// TwinCAT 3 PLC project Plc_Ampel
// ProgramVersion: 3.1.4023.0
// libraries:
//   Tc2_Standard, * (Beckhoff Automation GmbH)
//   Tc2_System, * (Beckhoff Automation GmbH)
//   Tc3_Module, * (Beckhoff Automation GmbH)
//   VisuSymbols,3.5.10.0,System
// project tree:
//   DUTs/ EN_TRAFFICLIGHT_STATE.TcDUT
//   / GlobalTextList.TcGTLO, PlcTask.TcTTO, Visualization Manager.TcVMO (not stored)
//   POUs/ MAIN.TcPOU, FB_TrafficLight.TcPOU
//   VISUs/ VISU_TrafficLight.TcVIS
// (motion and I/O tree: see PLC project plc_safe)
// real-time tasks:
//   TASK PlcTask: cycle T#10ms, priority 20, ADS port 350
//   TASK PlcTask1: cycle T#10ms, priority 21, ADS port 351

CONFIGURATION Plc_Ampel
    RESOURCE PLC ON TwinCAT3
        TASK PlcTask(INTERVAL := T#10ms, PRIORITY := 21);
        PROGRAM MAIN WITH PlcTask : MAIN;
    END_RESOURCE
END_CONFIGURATION

// ---- DUTs/EN_TRAFFICLIGHT_STATE.TcDUT
{attribute 'qualified_only'}
{attribute 'strict'}
TYPE EN_TRAFFICLIGHT_STATE :
(
	STATE_UNDEFINED := 0,
	STATE_INIT,
	STATE_DISABLED,
	STATE_RED,
	STATE_RED_YELLOW,
	STATE_YELLOW,
	STATE_GREEN
);
END_TYPE

// ---- POUs/MAIN.TcPOU
PROGRAM MAIN
VAR
	trafficLight_1			: FB_TrafficLight;
	
	// control variables
	clear					: BOOL;
	block					: BOOL;
	disable					: BOOL;
	
	// output variables
	red						: BOOL;
	yellow					: BOOL;
	green					: BOOL;
END_VAR

trafficLight_1(clear_road := clear, block_road := block, disable_system := disable);

red := trafficLight_1.red_light;
yellow := trafficLight_1.yellow_light;
green := trafficLight_1.green_light;

END_PROGRAM

// ---- POUs/FB_TrafficLight.TcPOU
FUNCTION_BLOCK FB_TrafficLight
VAR_INPUT
	clear_road 			: BOOL;
	block_road 			: BOOL;
	disable_system		: BOOL;
END_VAR
VAR_OUTPUT
	red_light			: BOOL;
	yellow_light		: BOOL;
	green_light			: BOOL;
END_VAR
VAR
	// state variables
	currentState		: 	EN_TRAFFICLIGHT_STATE := EN_TRAFFICLIGHT_STATE.STATE_INIT;
	lastState			: 	EN_TRAFFICLIGHT_STATE := EN_TRAFFICLIGHT_STATE.STATE_UNDEFINED;
	timer				: 	TON;
	// flag to reset the timer after the state machine has used it
	resetTimer			:	BOOL;
	// flag to update last state
	transitionDone		: 	BOOL;
END_VAR

timer();  // call timer

// state machine
CASE currentState OF
	EN_TRAFFICLIGHT_STATE.STATE_UNDEFINED:
	// jump to init	
	currentState := EN_TRAFFICLIGHT_STATE.STATE_INIT;
	
	//*****************************//
	EN_TRAFFICLIGHT_STATE.STATE_INIT:
	// jump to red
	currentState := EN_TRAFFICLIGHT_STATE.STATE_RED;
	
	//*****************************//
	EN_TRAFFICLIGHT_STATE.STATE_RED:
	// entry action
	IF(currentState <> lastState) THEN
		// enable only red light
		red_light := TRUE; yellow_light := FALSE; green_light := FALSE;
		lastState := currentState;  // update last state
	END_IF
	
	// clear road (prio 2)
	IF(clear_road) THEN
		currentState := EN_TRAFFICLIGHT_STATE.STATE_RED_YELLOW;
	END_IF
	
	// clear road (prio 1)
	IF(disable_system) THEN
		currentState := EN_TRAFFICLIGHT_STATE.STATE_DISABLED;
	END_IF
	
	//*****************************//
	EN_TRAFFICLIGHT_STATE.STATE_RED_YELLOW:
	// entry action
	IF(currentState <> lastState) THEN
		// enable red and yellow light
		red_light := TRUE; yellow_light := TRUE; green_light := FALSE;
		lastState := currentState;  // update last state
	END_IF
	
	// start timer for automatic state change
	timer.PT := T#2S;
	timer.IN := TRUE;
	
	// timer finished => exit action
	IF timer.Q THEN
		currentState := EN_TRAFFICLIGHT_STATE.STATE_GREEN;
		resetTimer := TRUE;
	END_IF
	
	//*****************************//
	EN_TRAFFICLIGHT_STATE.STATE_YELLOW:
	// entry action
	IF(currentState <> lastState) THEN
		// enable yellow light only
		red_light := FALSE; yellow_light := TRUE; green_light := FALSE;
		lastState := currentState;  // update last state
	END_IF
	
	// start timer for automatic state change
	timer.PT := T#5S;
	timer.IN := TRUE;
	
	// timer finished => exit action
	IF timer.Q THEN
		currentState := EN_TRAFFICLIGHT_STATE.STATE_RED;
		resetTimer := TRUE;
	END_IF
	
	//*****************************//
	EN_TRAFFICLIGHT_STATE.STATE_GREEN:
	// entry action
	IF(currentState <> lastState) THEN
		// enable green light only
		red_light := FALSE; yellow_light := FALSE; green_light := TRUE;
		lastState := currentState;  // update last state
	END_IF
	
	// block_road signal
	IF(block_road) THEN
		currentState := EN_TRAFFICLIGHT_STATE.STATE_YELLOW;
	END_IF
	
	//*****************************//
	EN_TRAFFICLIGHT_STATE.STATE_DISABLED:
	// disable all lights
	red_light := FALSE; green_light := FALSE;
	
	// start timer for yellow blinking
	timer.PT := T#1S;
	timer.IN := TRUE;
	
	// invert yellow light (blink)
	IF timer.Q THEN
		yellow_light := NOT yellow_light;
		resetTimer := TRUE;
	END_IF
	
	// system was re-enabled 
	IF (disable_system = FALSE) THEN
		lastState := currentState;  // update last state
		currentState := EN_TRAFFICLIGHT_STATE.STATE_RED;
		resetTimer := TRUE;
	END_IF
	
END_CASE

// reset timer since it was used
IF resetTimer THEN
	timer.IN := FALSE;
	timer();  // call to trigger edge
	resetTimer := FALSE;	
END_IF

END_FUNCTION_BLOCK

// ---- GlobalTextList.TcGTLO
TEXTLIST GlobalTextList
  241 = 'Block road'
  918 = 'Clear road'
  437 = 'Control'
  462 = 'Disable system'
  422 = 'Traffic Light'
END_TEXTLIST

// ---- VISUs/VISU_TrafficLight.TcVIS
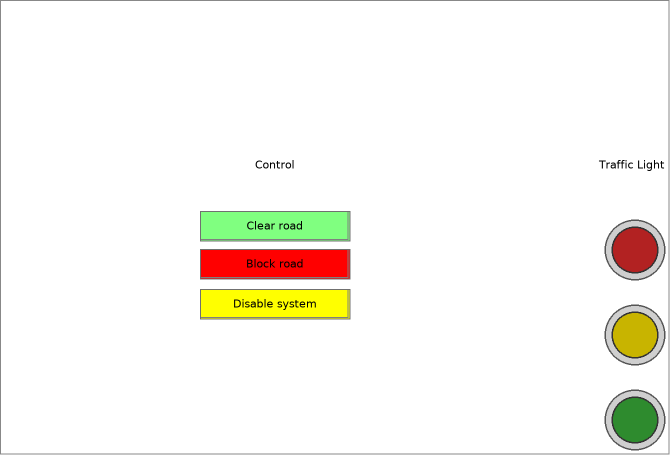
VISUALIZATION VISU_TrafficLight  // 670x455
    Button (200,211 150x30), "Clear road"
        tap MAIN.clear
    Button (200,249 150x30), "Block road"
        tap MAIN.block
    Button (200,289 150x30), "Disable system"
        toggle MAIN.disable
    Lamp1 (600,215 70x70), variable: MAIN.red, style: Lamp-Lamp1-Red
    Lamp1 (600,300 70x70), variable: MAIN.yellow, style: Lamp-Lamp1-Yellow
    Lamp1 (600,385 70x70), variable: MAIN.green, style: Lamp-Lamp1-Green
    Label (600,150 64x30), "Traffic Light"
    Label (200,150 150x30), "Control"
END_VISUALIZATION
